INTERFACE I_TemperatureSensor

METHOD Run
VAR_INPUT
END_VAR
END_METHOD

PROPERTY Temperature : REAL
GET
END_GET
SET
END_SET
END_PROPERTY

END_INTERFACE

(* stored: Version 1.1.0.1, ProductVersion 3.1.4024.0
   Itf I_TemperatureSensor: Id {49488df3-dbfc-4e57-b26b-56381a9ee01b}
   Method Run: Id {a887ec2b-5ded-41e4-a836-d66d8f3ae003}
   Property Temperature: Id {0feb6fe9-d9b1-42f8-8eb2-f000fe631ab0}
   Get Get: Id {e3763511-b0c7-46f5-a86a-b9fe34f56290}
   Set Set: Id {8660d4b4-18bc-414d-9032-d035388a320a} *)
